ABB RobotStudio station: HuiswerkOpdrachten.rsstnx

Station HuiswerkOpdrachten (saved by RobotStudio 23.3.10550.0)
Controller IRB120FGL_3_58
  mechanical unit ROB_1: IRB120FGL_3_58__01, 6 joints, base frame (0, 0, 0) mm
Layout (positions relative to the parent item):
  - IRB120FGL_3_58__01 [mechanism, from %ABB.RobotStudio.Models.IRB120%\IRB120FGL_3_58__01.rslib] at (0, 0, 0) mm; joint values [0, 0, 0, 0, 0.5236, 0] (rad or m)
Targets, tools, work objects and paths stored in the station, written as RAPID:
! task T_ROB1
MODULE MainModule
  CONST robtarget Target_10:=[[-0.000012646,-289.300007188,499.999964135],[0,0,1,0.000000007],[-2,-1,-2,0],[9E+09,9E+09,9E+09,9E+09,9E+09,9E+09]];
  CONST jointtarget JointTarget_3:=[[0,0,0,0,0,0],[9E+09,9E+09,9E+09,9E+09,9E+09,9E+09]];
  PROC Path_10()
    MoveJ Target_10,v1000,z100,tool0\WObj:=wobj0;
  ENDPROC
ENDMODULE

